// Mitsubishi GX Works2 project: BookEX6_34 DataProcess   PLC: Q13UDV

// global labels: Global
VAR_GLOBAL
  bVar0 AT M5000 : BOOL;
  abArray0 AT M5010 : ARRAY [0..49] OF BOOL;
  sStr0 AT D5000 : STRING[199];
  sStr1 AT D5100 : STRING[199];
  sStr2 AT D5200 : STRING[199];
  sStr3 AT D5300 : STRING[199];
  sStr4 AT D5400 : STRING[199];
  sStr5 AT D5500 : STRING[199];
  sStr6 AT D5600 : STRING[199];
  sStr7 AT D5700 : STRING[199];
  sStr8 AT D5800 : STRING[199];
  sStr9 AT D5900 : STRING[199];
  iVar0 AT D4500 : INT;
  iVar1 AT D4501 : INT;
  iVar2 AT D4502 : INT;
  iVar3 AT D4503 : INT;
  iVar4 AT D4504 : INT;
  iVar5 AT D4505 : INT;
  iVar6 AT D4506 : INT;
  iVar7 AT D4507 : INT;
  iVar8 AT D4508 : INT;
  iVar9 AT D4509 : INT;
  dVar0 AT D4510 : DINT;
  dVar1 AT D4512 : DINT;
  dVar2 AT D4514 : DINT;
  dVar3 AT D4516 : DINT;
  dVar4 AT D4518 : DINT;
  dVar5 AT D4520 : DINT;
  dVar6 AT D4522 : DINT;
  dVar7 AT D4524 : DINT;
  dVar8 AT D4526 : DINT;
  dVar9 AT D4528 : DINT;
  wVar0 AT D4530 : WORD;
  wVar1 AT D4531 : WORD;
  wVar2 AT D4532 : WORD;
  wVar3 AT D4533 : WORD;
  wVar4 AT D4534 : WORD;
  wVar5 AT D4535 : WORD;
  wVar6 AT D4536 : WORD;
  wVar7 AT D4537 : WORD;
  wVar8 AT D4538 : WORD;
  wVar9 AT D4539 : WORD;
  dwVar0 AT D4540 : DWORD;
  dwVar1 AT D4542 : DWORD;
  dwVar2 AT D4544 : DWORD;
  dwVar3 AT D4546 : DWORD;
  dwVar4 AT D4548 : DWORD;
  dwVar5 AT D4550 : DWORD;
  dwVar6 AT D4552 : DWORD;
  dwVar7 AT D4554 : DWORD;
  dwVar8 AT D4556 : DWORD;
  dwVar9 AT D4558 : DWORD;
  fsVar0 AT D4560 : REAL;
  fsVar1 AT D4562 : REAL;
  fsVar2 AT D4564 : REAL;
  fsVar3 AT D4566 : REAL;
  fsVar4 AT D4568 : REAL;
  fsVar5 AT D4570 : REAL;
  fsVar6 AT D4572 : REAL;
  fsVar7 AT D4574 : REAL;
  fsVar8 AT D4576 : REAL;
  fsVar9 AT D4578 : REAL;
  fdVar0 AT D4580 : LREAL;
  tTime0 AT D4620 : TIME;
  tTime1 AT D4622 : TIME;
  tTime2 AT D4624 : TIME;
  tTime3 AT D4626 : TIME;
  tTime4 AT D4628 : TIME;
  tTime5 AT D4630 : TIME;
  tTime6 AT D4632 : TIME;
  tTime7 AT D4634 : TIME;
  tTime8 AT D4636 : TIME;
  tTime9 AT D4638 : TIME;
  tTime10 AT D4640 : TIME;
  bVar1 AT M5001 : BOOL;
  bVar2 AT M5002 : BOOL;
  bVar3 AT M5003 : BOOL;
  bVar4 AT M5004 : BOOL;
  bVar5 AT M5005 : BOOL;
  bVar6 AT M5006 : BOOL;
  bVar7 AT M5007 : BOOL;
  bVar8 AT M5008 : BOOL;
  bVar9 AT M5009 : BOOL;
  abArray1 AT M5060 : ARRAY [0..49] OF BOOL;
  abArray2 AT M5110 : ARRAY [0..49] OF BOOL;
  abArray3 AT M5160 : ARRAY [0..49] OF BOOL;
  abArray4 AT M5210 : ARRAY [0..49] OF BOOL;
  abArray5 AT M5260 : ARRAY [0..49] OF BOOL;
  abArray6 AT M5310 : ARRAY [0..49] OF BOOL;
  abArray7 AT M5360 : ARRAY [0..49] OF BOOL;
  abArray8 AT M5410 : ARRAY [0..49] OF BOOL;
  abArray9 AT M5460 : ARRAY [0..49] OF BOOL;
  fdVar1 AT D4584 : LREAL;
  fdVar2 AT D4588 : LREAL;
  fdVar3 AT D4592 : LREAL;
  fdVar4 AT D4596 : LREAL;
  fdVar5 AT D4600 : LREAL;
  fdVar6 AT D4604 : LREAL;
  fdVar7 AT D4608 : LREAL;
  fdVar8 AT D4612 : LREAL;
  fdVar9 AT D4616 : LREAL;
  afsPen0 AT D2000 : ARRAY [0..499] OF REAL;
  afsPen1 AT D3000 : ARRAY [0..499] OF REAL;
END_VAR
// user libraries (not included): HMI

PROGRAM ExCCD
VAR
  aiVar8 : ARRAY [0..1] OF INT;
  aiVar16 : ARRAY [0..1] OF INT;
END_VAR
(* structured ladder/FBD written out as ST: instructions are called as NAME(EN, inputs, outputs); _pN, _eN, _tN stand for wires *)
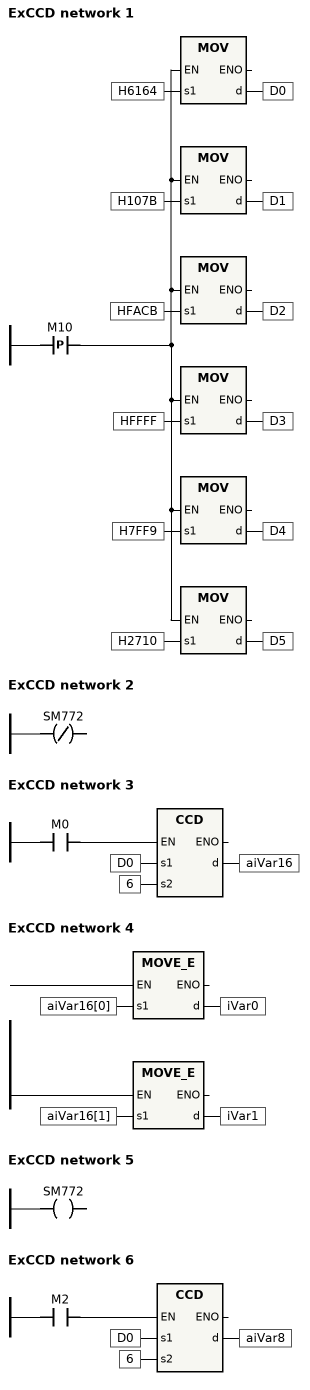
(* network 1 *)
_p1 := LDP(TRUE, M10);
MOV(_p1, H6164, D0);
MOV(_p1, H107B, D1);
MOV(_p1, HFACB, D2);
MOV(_p1, HFFFF, D3);
MOV(_p1, H7FF9, D4);
MOV(_p1, H2710, D5);
(* network 2 *)
SM772 := NOT TRUE;
(* network 3 *)
CCD(M0, D0, 6, aiVar16);
(* network 4 *)
MOVE_E(TRUE, aiVar16[0], iVar0);
MOVE_E(TRUE, aiVar16[1], iVar1);
(* network 5 *)
SM772 := TRUE;
(* network 6 *)
CCD(M2, D0, 6, aiVar8);
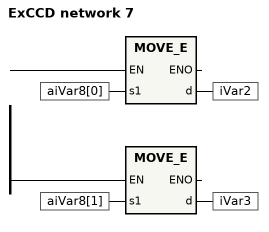
(* network 7 *)
MOVE_E(TRUE, aiVar8[0], iVar2);
MOVE_E(TRUE, aiVar8[1], iVar3);
END_PROGRAM

PROGRAM ExCRC
VAR
  aiVar0 : ARRAY [0..1] OF INT;
  aiVar1 : ARRAY [0..1] OF INT;
  aiVar2 : ARRAY [0..3] OF INT;
  aiVar3 : ARRAY [0..2] OF INT;
  Mov8INT_1 : Mov8INT;
  GetCRC_1 : GetCRC;
  GetCRC_2 : GetCRC;
END_VAR
(* structured ladder/FBD written out as ST: instructions are called as NAME(EN, inputs, outputs); _pN, _eN, _tN stand for wires *)
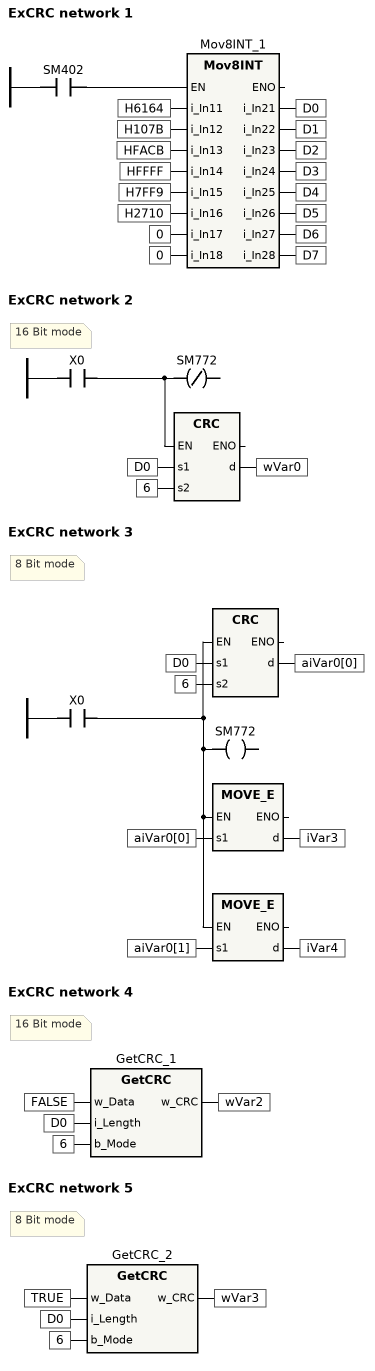
(* network 1 *)
Mov8INT_1(EN := SM402, i_In11 := H6164, i_In12 := H107B, i_In13 := HFACB, i_In14 := HFFFF, i_In15 := H7FF9, i_In16 := H2710, i_In17 := 0, i_In18 := 0, i_In21 => D0, i_In22 => D1, i_In23 => D2, i_In24 => D3, i_In25 => D4, i_In26 => D5, i_In27 => D6, i_In28 => D7);
(* network 2 *)
(* 16 Bit mode *)
SM772 := NOT X0;
CRC(X0, D0, 6, wVar0);
(* network 3 *)
(* 8 Bit mode *)
SM772 := X0;
CRC(X0, D0, 6, aiVar0[0]);
MOVE_E(X0, aiVar0[0], iVar3);
MOVE_E(X0, aiVar0[1], iVar4);
(* network 4 *)
(* 16 Bit mode *)
GetCRC_1(w_Data := FALSE, i_Length := D0, b_Mode := 6, w_CRC => wVar2);
(* network 5 *)
(* 8 Bit mode *)
GetCRC_2(w_Data := TRUE, i_Length := D0, b_Mode := 6, w_CRC => wVar3);
END_PROGRAM

PROGRAM ExDECO
VAR
  abArr0 : ARRAY [0..2] OF BOOL;
  Decode8_1 : Decode8;
  abArr1 : ARRAY [0..7] OF BOOL;
  Decode4_1 : Decode4;
  Decode8_2 : Decode8;
  bMan : BOOL;
  bSemi : BOOL;
  bAuto : BOOL;
  bMaint : BOOL;
END_VAR
(* structured ladder/FBD written out as ST: instructions are called as NAME(EN, inputs, outputs); _pN, _eN, _tN stand for wires *)
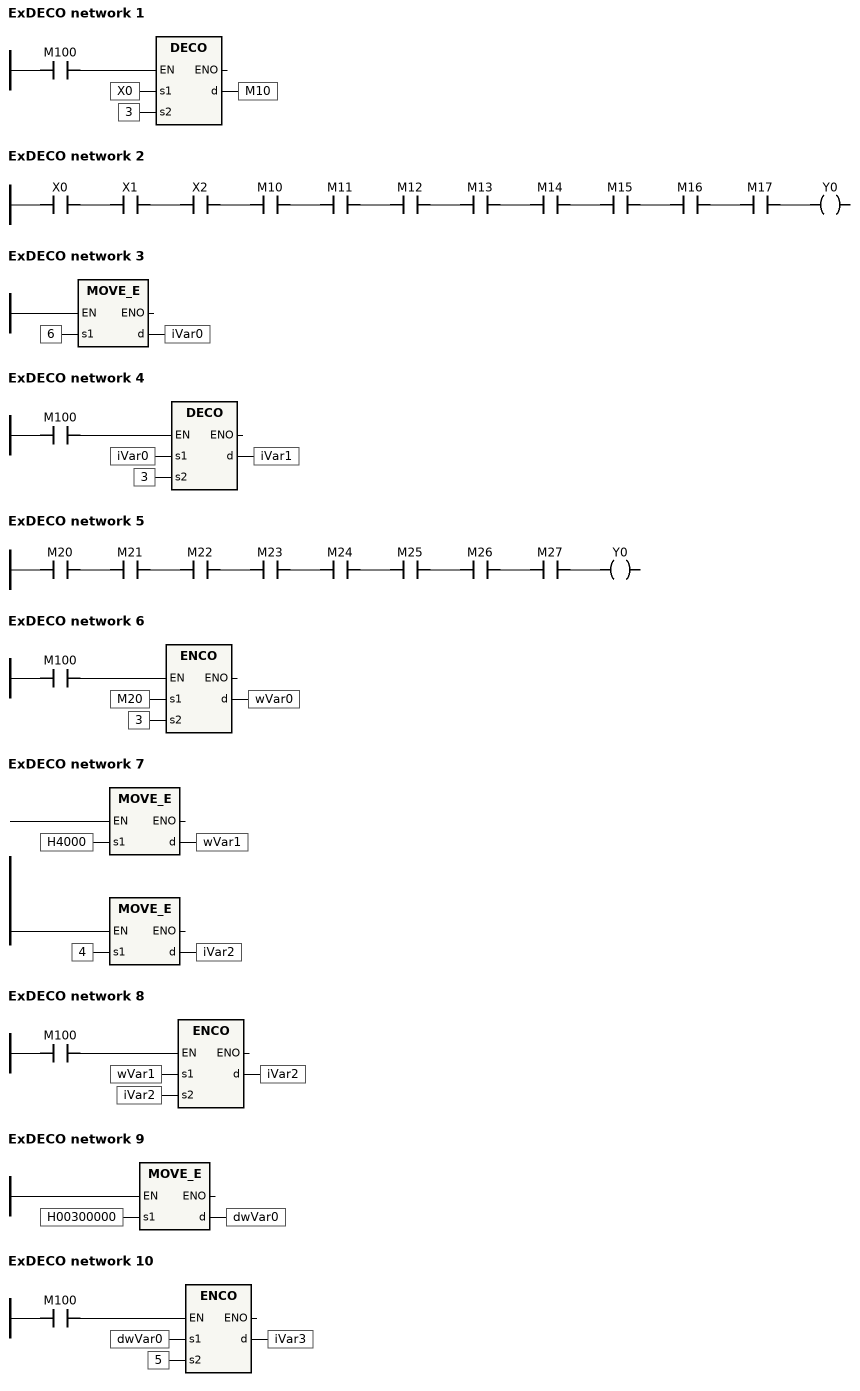
(* network 1 *)
DECO(M100, X0, 3, M10);
(* network 2 *)
Y0 := X0 AND X1 AND X2 AND M10 AND M11 AND M12 AND M13 AND M14 AND M15 AND M16 AND M17;
(* network 3 *)
MOVE_E(TRUE, 6, iVar0);
(* network 4 *)
DECO(M100, iVar0, 3, iVar1);
(* network 5 *)
Y0 := M20 AND M21 AND M22 AND M23 AND M24 AND M25 AND M26 AND M27;
(* network 6 *)
ENCO(M100, M20, 3, wVar0);
(* network 7 *)
MOVE_E(TRUE, H4000, wVar1);
MOVE_E(TRUE, 4, iVar2);
(* network 8 *)
ENCO(M100, wVar1, iVar2, iVar2);
(* network 9 *)
MOVE_E(TRUE, H00300000, dwVar0);
(* network 10 *)
ENCO(M100, dwVar0, 5, iVar3);
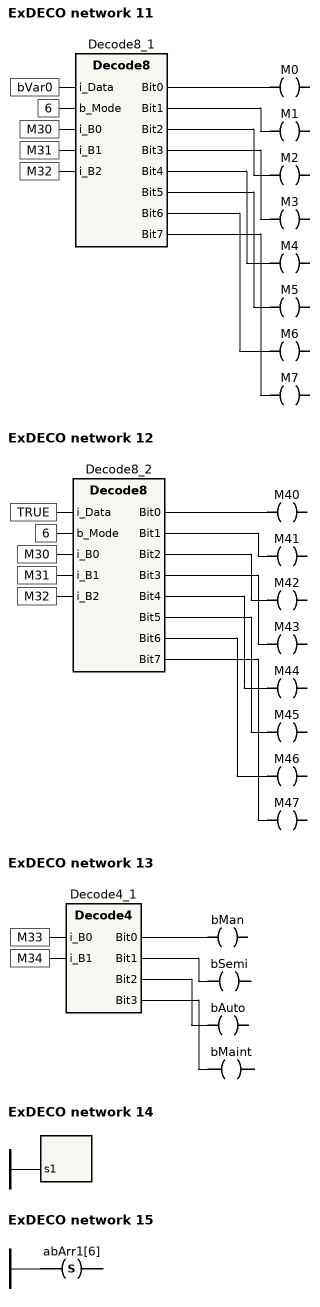
(* network 11 *)
Decode8_1(i_Data := bVar0, b_Mode := 6, i_B0 := M30, i_B1 := M31, i_B2 := M32);
M0 := Decode8_1.Bit0;
M1 := Decode8_1.Bit1;
M2 := Decode8_1.Bit2;
M3 := Decode8_1.Bit3;
M4 := Decode8_1.Bit4;
M5 := Decode8_1.Bit5;
M6 := Decode8_1.Bit6;
M7 := Decode8_1.Bit7;
(* network 12 *)
Decode8_2(i_Data := TRUE, b_Mode := 6, i_B0 := M30, i_B1 := M31, i_B2 := M32);
M40 := Decode8_2.Bit0;
M41 := Decode8_2.Bit1;
M42 := Decode8_2.Bit2;
M43 := Decode8_2.Bit3;
M44 := Decode8_2.Bit4;
M45 := Decode8_2.Bit5;
M46 := Decode8_2.Bit6;
M47 := Decode8_2.Bit7;
(* network 13 *)
Decode4_1(i_B0 := M33, i_B1 := M34);
bMan := Decode4_1.Bit0;
bSemi := Decode4_1.Bit1;
bAuto := Decode4_1.Bit2;
bMaint := Decode4_1.Bit3;
(* network 14 *)
(* element kind 10  <- TRUE *)
(* network 15 *)
SET(TRUE, abArr1[6]);
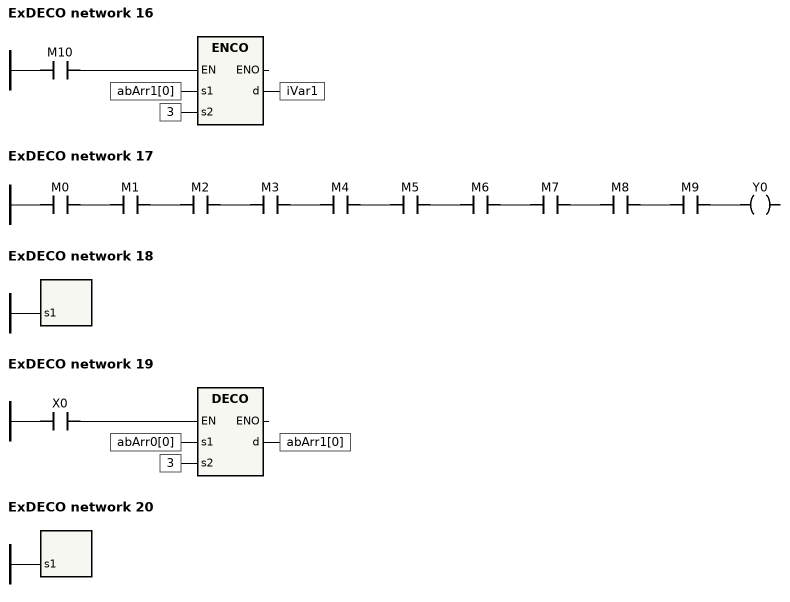
(* network 16 *)
ENCO(M10, abArr1[0], 3, iVar1);
(* network 17 *)
Y0 := M0 AND M1 AND M2 AND M3 AND M4 AND M5 AND M6 AND M7 AND M8 AND M9;
(* network 18 *)
(* element kind 10  <- TRUE *)
(* network 19 *)
DECO(X0, abArr0[0], 3, abArr1[0]);
(* network 20 *)
(* element kind 10  <- TRUE *)
END_PROGRAM

PROGRAM ExDIS
VAR
  Mov4WORD_1 : Mov4WORD;
  DDIS_1 : DDIS;
END_VAR
(* structured ladder/FBD written out as ST: instructions are called as NAME(EN, inputs, outputs); _pN, _eN, _tN stand for wires *)
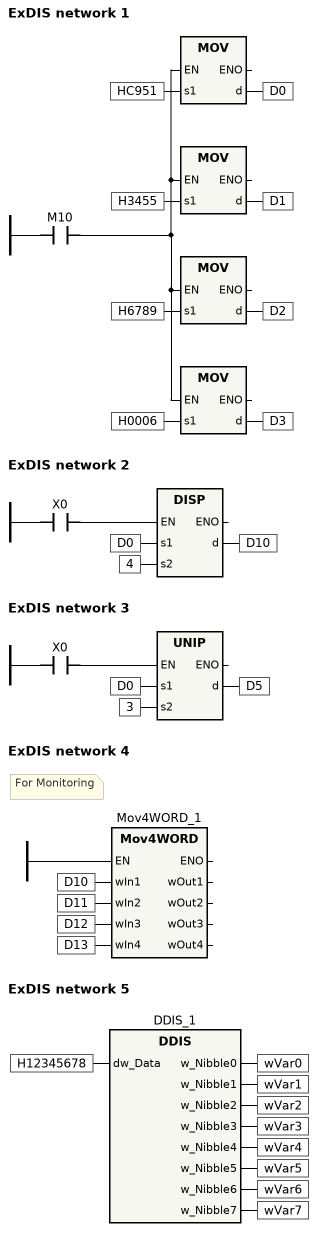
(* network 1 *)
MOV(M10, HC951, D0);
MOV(M10, H3455, D1);
MOV(M10, H6789, D2);
MOV(M10, H0006, D3);
(* network 2 *)
DISP(X0, D0, 4, D10);
(* network 3 *)
UNIP(X0, D0, 3, D5);
(* network 4 *)
(* For Monitoring *)
Mov4WORD_1(EN := TRUE, wIn1 := D10, wIn2 := D11, wIn3 := D12, wIn4 := D13);
(* network 5 *)
DDIS_1(dw_Data := H12345678, w_Nibble0 => wVar0, w_Nibble1 => wVar1, w_Nibble2 => wVar2, w_Nibble3 => wVar3, w_Nibble4 => wVar4, w_Nibble5 => wVar5, w_Nibble6 => wVar6, w_Nibble7 => wVar7);
END_PROGRAM

PROGRAM ExGetParity
VAR
  GetParity_1 : GetParity;
  awTestData : ARRAY [0..255] OF WORD;
  GetParity_2 : GetParity;
END_VAR
(* structured ladder/FBD written out as ST: instructions are called as NAME(EN, inputs, outputs); _pN, _eN, _tN stand for wires *)
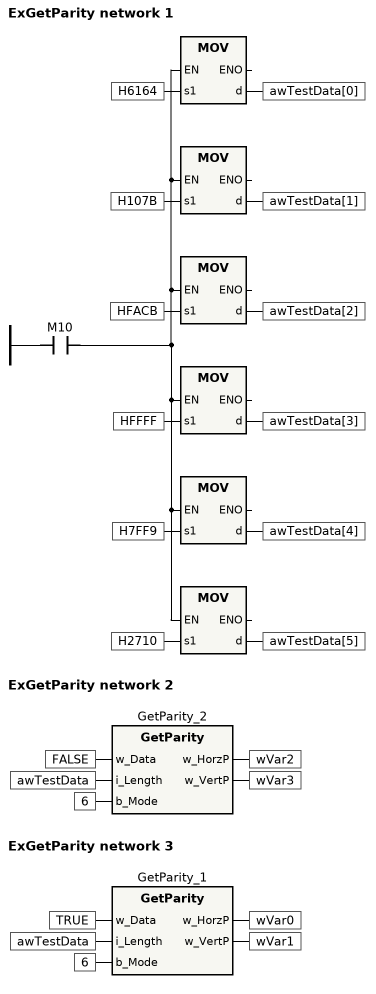
(* network 1 *)
MOV(M10, H6164, awTestData[0]);
MOV(M10, H107B, awTestData[1]);
MOV(M10, HFACB, awTestData[2]);
MOV(M10, HFFFF, awTestData[3]);
MOV(M10, H7FF9, awTestData[4]);
MOV(M10, H2710, awTestData[5]);
(* network 2 *)
GetParity_2(w_Data := FALSE, i_Length := awTestData, b_Mode := 6, w_HorzP => wVar2, w_VertP => wVar3);
(* network 3 *)
GetParity_1(w_Data := TRUE, i_Length := awTestData, b_Mode := 6, w_HorzP => wVar0, w_VertP => wVar1);
END_PROGRAM

PROGRAM ExMAX
VAR
  Mov4WORD_1 : Mov4WORD;
  Mov4WORD_2 : Mov4WORD;
  Mov4WORD_3 : Mov4WORD;
  dVa : ARRAY [0..1] OF DINT;
  RealMIN_MAX_1 : RealMIN_MAX;
  afsData : ARRAY [0..31] OF REAL;
END_VAR
(* structured ladder/FBD written out as ST: instructions are called as NAME(EN, inputs, outputs); _pN, _eN, _tN stand for wires *)
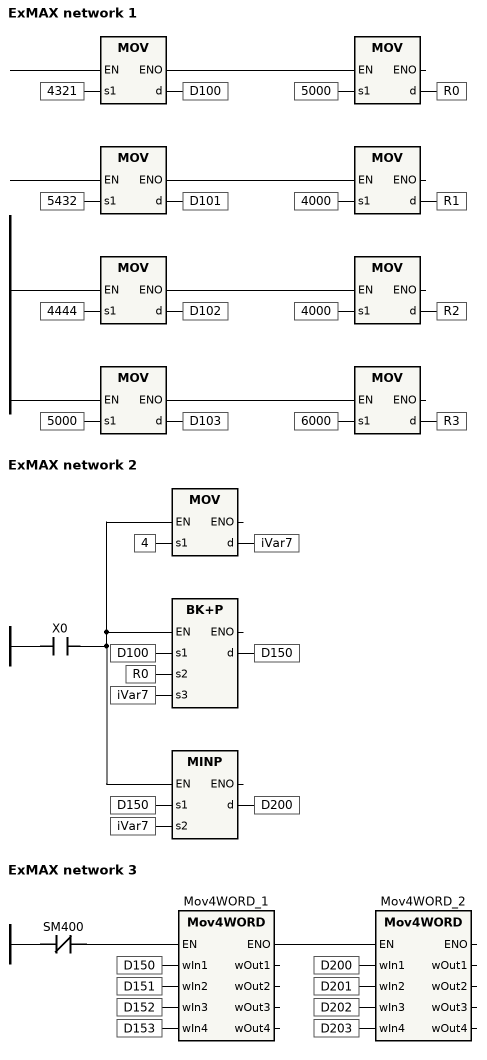
(* network 1 *)
_e1 := MOV(TRUE, 4321, D100);
MOV(_e1, 5000, R0);
_e2 := MOV(TRUE, 5432, D101);
MOV(_e2, 4000, R1);
_e3 := MOV(TRUE, 4444, D102);
MOV(_e3, 4000, R2);
_e4 := MOV(TRUE, 5000, D103);
MOV(_e4, 6000, R3);
(* network 2 *)
MOV(X0, 4, iVar7);
BK+P(X0, D100, R0, iVar7, D150);
MINP(X0, D150, iVar7, D200);
(* network 3 *)
Mov4WORD_1(EN := NOT SM400, wIn1 := D150, wIn2 := D151, wIn3 := D152, wIn4 := D153);
Mov4WORD_2(EN := Mov4WORD_1.ENO, wIn1 := D200, wIn2 := D201, wIn3 := D202, wIn4 := D203);
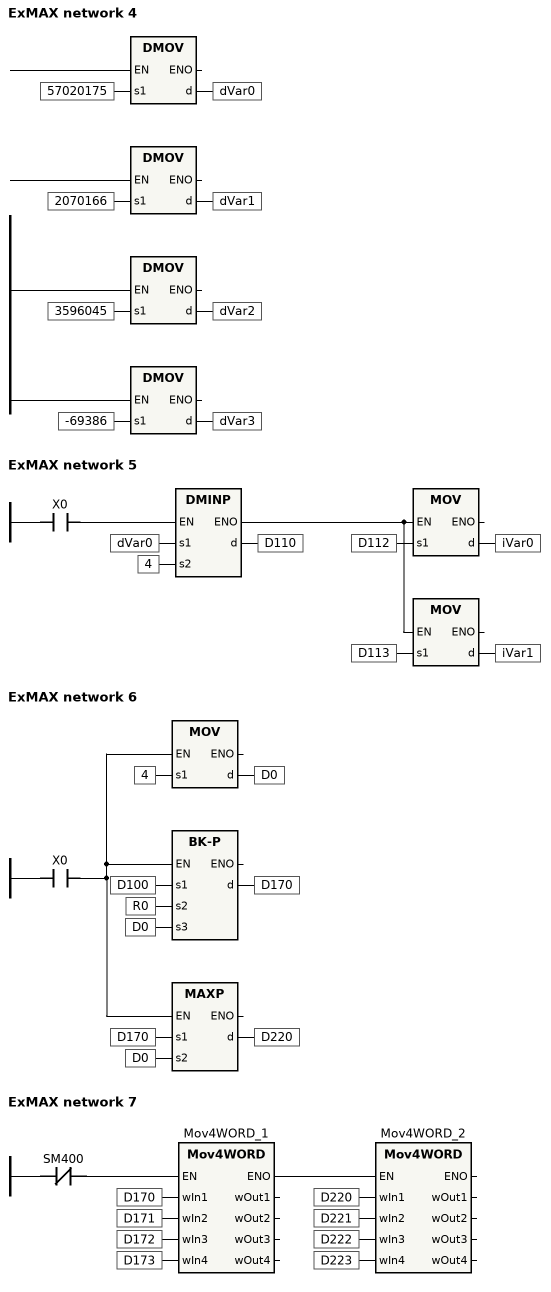
(* network 4 *)
DMOV(TRUE, 57020175, dVar0);
DMOV(TRUE, 2070166, dVar1);
DMOV(TRUE, 3596045, dVar2);
DMOV(TRUE, -69386, dVar3);
(* network 5 *)
_e1 := DMINP(X0, dVar0, 4, D110);
MOV(_e1, D112, iVar0);
MOV(_e1, D113, iVar1);
(* network 6 *)
MOV(X0, 4, D0);
BK-P(X0, D100, R0, D0, D170);
MAXP(X0, D170, D0, D220);
(* network 7 *)
Mov4WORD_1(EN := NOT SM400, wIn1 := D170, wIn2 := D171, wIn3 := D172, wIn4 := D173);
Mov4WORD_2(EN := Mov4WORD_1.ENO, wIn1 := D220, wIn2 := D221, wIn3 := D222, wIn4 := D223);
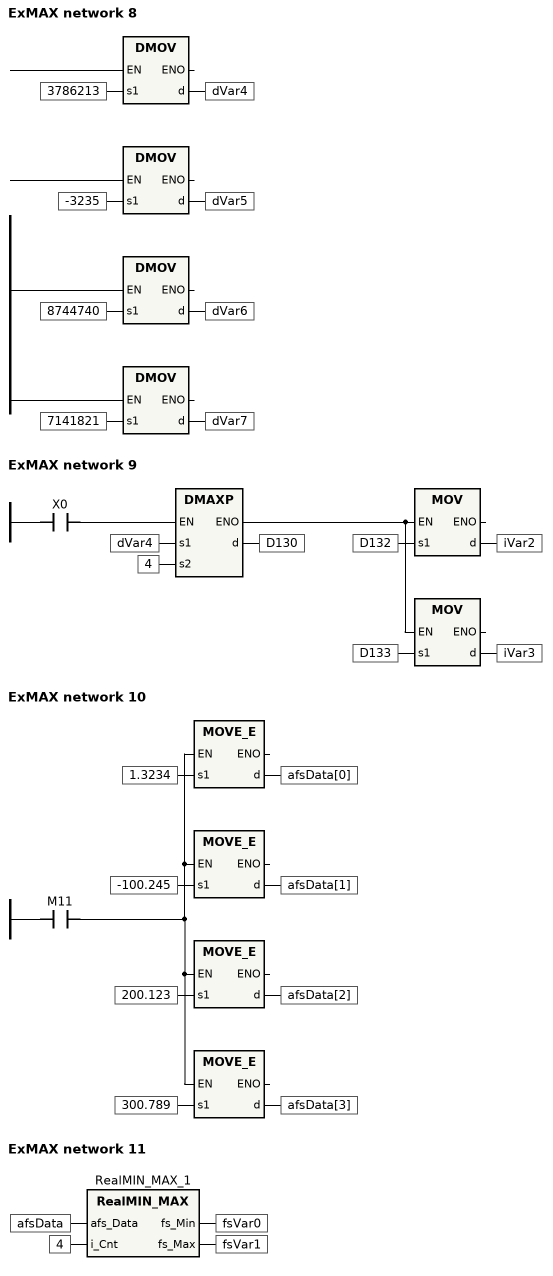
(* network 8 *)
DMOV(TRUE, 3786213, dVar4);
DMOV(TRUE, -3235, dVar5);
DMOV(TRUE, 8744740, dVar6);
DMOV(TRUE, 7141821, dVar7);
(* network 9 *)
_e1 := DMAXP(X0, dVar4, 4, D130);
MOV(_e1, D132, iVar2);
MOV(_e1, D133, iVar3);
(* network 10 *)
MOVE_E(M11, 1.3234, afsData[0]);
MOVE_E(M11, -100.245, afsData[1]);
MOVE_E(M11, 200.123, afsData[2]);
MOVE_E(M11, 300.789, afsData[3]);
(* network 11 *)
RealMIN_MAX_1(afs_Data := afsData, i_Cnt := 4, fs_Min => fsVar0, fs_Max => fsVar1);
END_PROGRAM

PROGRAM ExMEAN
VAR
  afsData : ARRAY [0..31] OF REAL;
END_VAR
(* structured ladder/FBD written out as ST: instructions are called as NAME(EN, inputs, outputs); _pN, _eN, _tN stand for wires *)
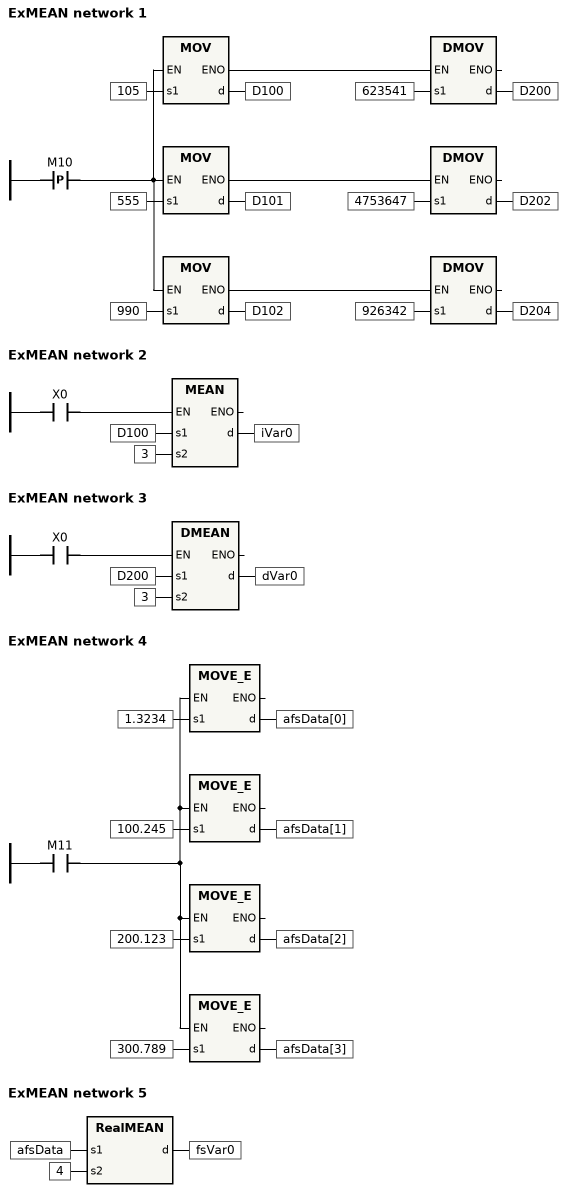
(* network 1 *)
_p1 := LDP(TRUE, M10);
_e2 := MOV(_p1, 105, D100);
DMOV(_e2, 623541, D200);
_e3 := MOV(_p1, 555, D101);
DMOV(_e3, 4753647, D202);
_e4 := MOV(_p1, 990, D102);
DMOV(_e4, 926342, D204);
(* network 2 *)
MEAN(X0, D100, 3, iVar0);
(* network 3 *)
DMEAN(X0, D200, 3, dVar0);
(* network 4 *)
MOVE_E(M11, 1.3234, afsData[0]);
MOVE_E(M11, 100.245, afsData[1]);
MOVE_E(M11, 200.123, afsData[2]);
MOVE_E(M11, 300.789, afsData[3]);
(* network 5 *)
fsVar0 := RealMEAN(afsData, 4);
END_PROGRAM

PROGRAM ExNDIS
VAR
  Mov4WORD_1 : Mov4WORD;
END_VAR
(* structured ladder/FBD written out as ST: instructions are called as NAME(EN, inputs, outputs); _pN, _eN, _tN stand for wires *)
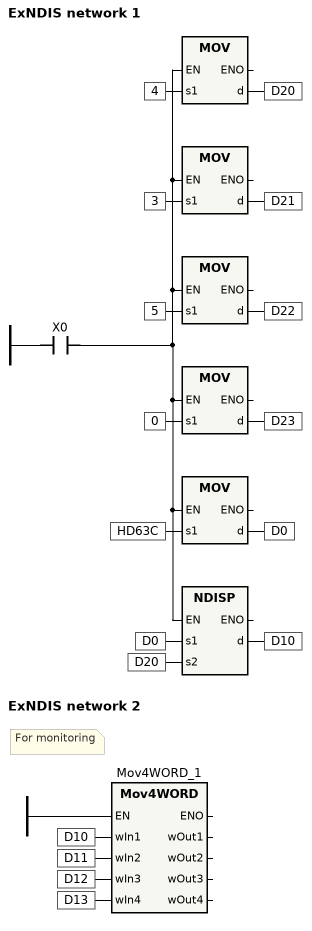
(* network 1 *)
MOV(X0, 4, D20);
MOV(X0, 3, D21);
MOV(X0, 5, D22);
MOV(X0, 0, D23);
MOV(X0, HD63C, D0);
NDISP(X0, D0, D20, D10);
(* network 2 *)
(* For monitoring *)
Mov4WORD_1(EN := TRUE, wIn1 := D10, wIn2 := D11, wIn3 := D12, wIn4 := D13);
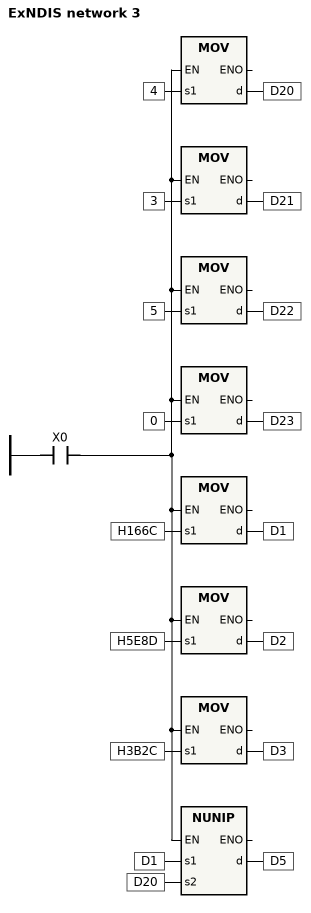
(* network 3 *)
MOV(X0, 4, D20);
MOV(X0, 3, D21);
MOV(X0, 5, D22);
MOV(X0, 0, D23);
MOV(X0, H166C, D1);
MOV(X0, H5E8D, D2);
MOV(X0, H3B2C, D3);
NUNIP(X0, D1, D20, D5);
END_PROGRAM

PROGRAM ExSearch
VAR
  Search_1 : Search;
  aiData : ARRAY [0..255] OF INT;
  DSearch_1 : DSearch;
  adData : ARRAY [0..255] OF DINT;
END_VAR
(* structured ladder/FBD written out as ST: instructions are called as NAME(EN, inputs, outputs); _pN, _eN, _tN stand for wires *)
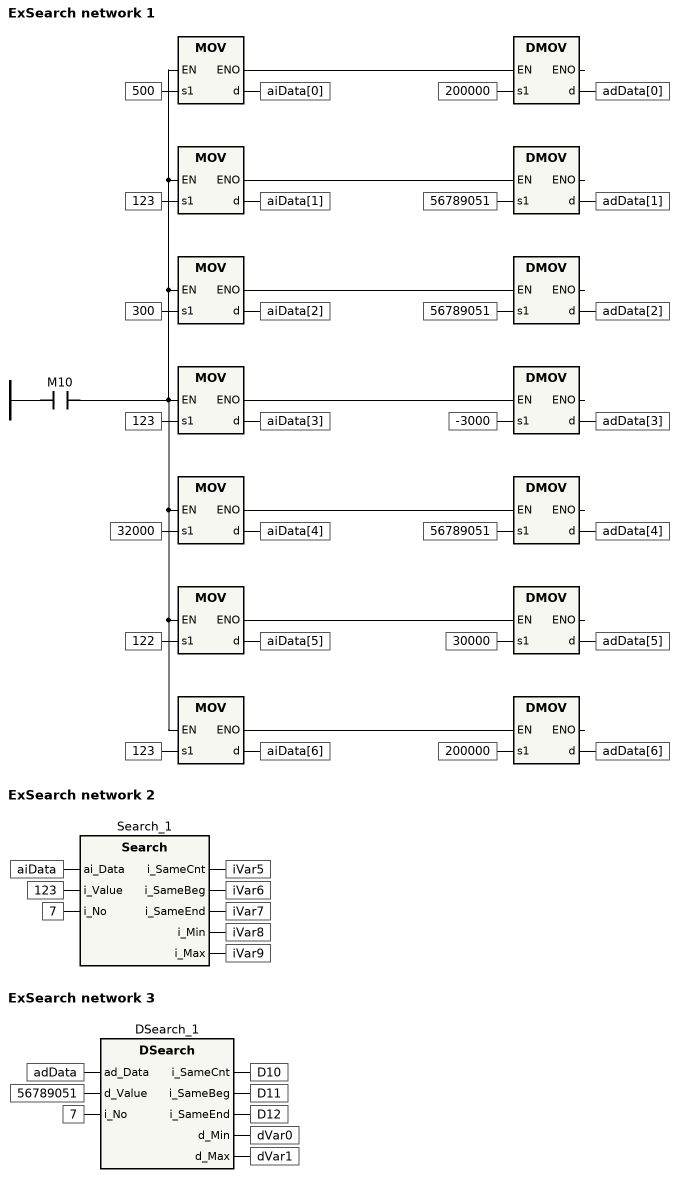
(* network 1 *)
_e1 := MOV(M10, 500, aiData[0]);
DMOV(_e1, 200000, adData[0]);
_e2 := MOV(M10, 123, aiData[1]);
DMOV(_e2, 56789051, adData[1]);
_e3 := MOV(M10, 300, aiData[2]);
DMOV(_e3, 56789051, adData[2]);
_e4 := MOV(M10, 123, aiData[3]);
DMOV(_e4, -3000, adData[3]);
_e5 := MOV(M10, 32000, aiData[4]);
DMOV(_e5, 56789051, adData[4]);
_e6 := MOV(M10, 122, aiData[5]);
DMOV(_e6, 30000, adData[5]);
_e7 := MOV(M10, 123, aiData[6]);
DMOV(_e7, 200000, adData[6]);
(* network 2 *)
Search_1(ai_Data := aiData, i_Value := 123, i_No := 7, i_SameCnt => iVar5, i_SameBeg => iVar6, i_SameEnd => iVar7, i_Min => iVar8, i_Max => iVar9);
(* network 3 *)
DSearch_1(ad_Data := adData, d_Value := 56789051, i_No := 7, i_SameCnt => D10, i_SameBeg => D11, i_SameEnd => D12, d_Min => dVar0, d_Max => dVar1);
END_PROGRAM

PROGRAM ExSEG
VAR
  aiClock : ARRAY [0..6] OF INT;
  aiMin : ARRAY [0..1] OF INT;
  aiSec : ARRAY [0..1] OF INT;
  aiHour : ARRAY [0..1] OF INT;
END_VAR
(* structured ladder/FBD written out as ST: instructions are called as NAME(EN, inputs, outputs); _pN, _eN, _tN stand for wires *)
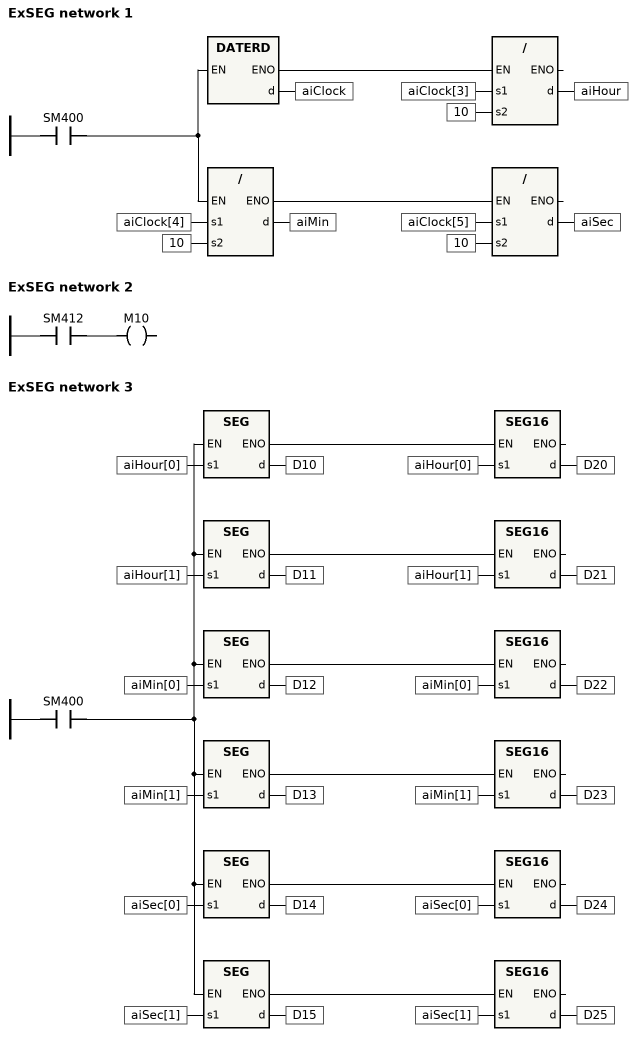
(* network 1 *)
_e1 := DATERD(SM400, aiClock);
/(_e1, aiClock[3], 10, aiHour);
_e2 := /(SM400, aiClock[4], 10, aiMin);
/(_e2, aiClock[5], 10, aiSec);
(* network 2 *)
M10 := SM412;
(* network 3 *)
_e1 := SEG(SM400, aiHour[0], D10);
SEG16(_e1, aiHour[0], D20);
_e2 := SEG(SM400, aiHour[1], D11);
SEG16(_e2, aiHour[1], D21);
_e3 := SEG(SM400, aiMin[0], D12);
SEG16(_e3, aiMin[0], D22);
_e4 := SEG(SM400, aiMin[1], D13);
SEG16(_e4, aiMin[1], D23);
_e5 := SEG(SM400, aiSec[0], D14);
SEG16(_e5, aiSec[0], D24);
_e6 := SEG(SM400, aiSec[1], D15);
SEG16(_e6, aiSec[1], D25);
END_PROGRAM

PROGRAM ExSER
VAR
  aiVar0 : ARRAY [0..1] OF INT;
  aiVar1 : ARRAY [0..1] OF INT;
  adVar0 : ARRAY [0..1] OF DINT;
  aiVar2 : ARRAY [0..3] OF INT;
  aiVar3 : ARRAY [0..2] OF INT;
END_VAR
(* structured ladder/FBD written out as ST: instructions are called as NAME(EN, inputs, outputs); _pN, _eN, _tN stand for wires *)
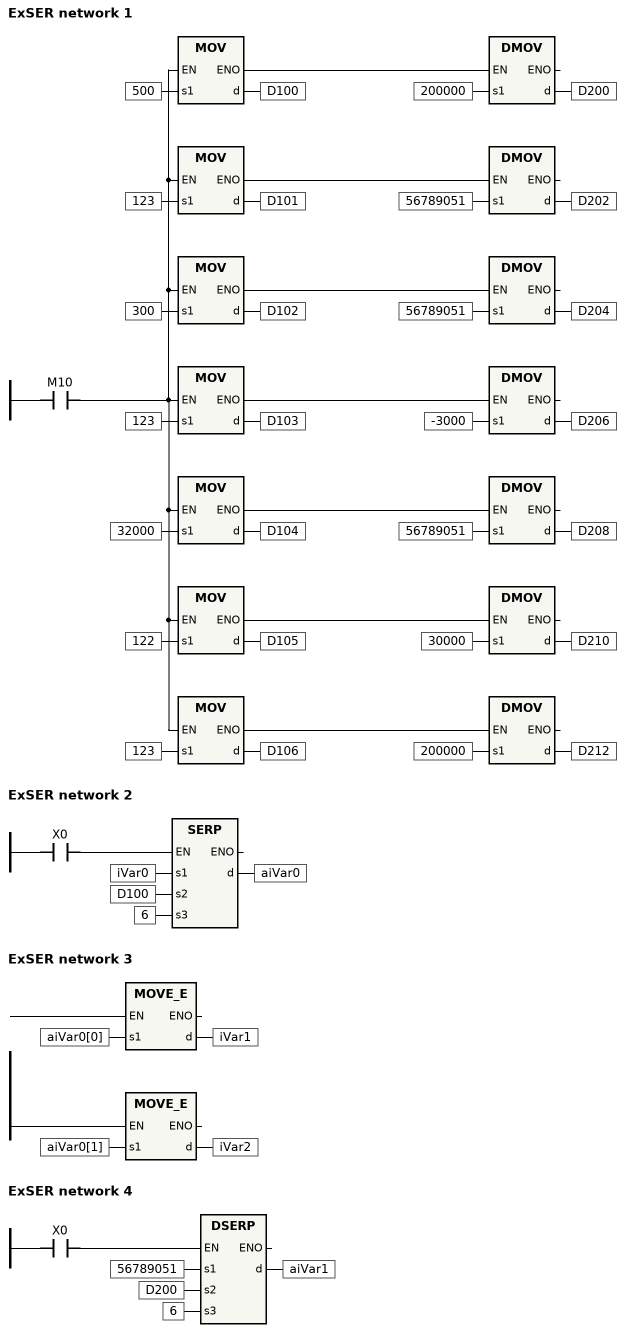
(* network 1 *)
_e1 := MOV(M10, 500, D100);
DMOV(_e1, 200000, D200);
_e2 := MOV(M10, 123, D101);
DMOV(_e2, 56789051, D202);
_e3 := MOV(M10, 300, D102);
DMOV(_e3, 56789051, D204);
_e4 := MOV(M10, 123, D103);
DMOV(_e4, -3000, D206);
_e5 := MOV(M10, 32000, D104);
DMOV(_e5, 56789051, D208);
_e6 := MOV(M10, 122, D105);
DMOV(_e6, 30000, D210);
_e7 := MOV(M10, 123, D106);
DMOV(_e7, 200000, D212);
(* network 2 *)
SERP(X0, iVar0, D100, 6, aiVar0);
(* network 3 *)
MOVE_E(TRUE, aiVar0[0], iVar1);
MOVE_E(TRUE, aiVar0[1], iVar2);
(* network 4 *)
DSERP(X0, 56789051, D200, 6, aiVar1);
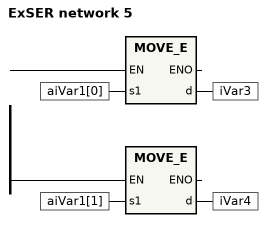
(* network 5 *)
MOVE_E(TRUE, aiVar1[0], iVar3);
MOVE_E(TRUE, aiVar1[1], iVar4);
END_PROGRAM

PROGRAM EXSORT
VAR
  SortBubble_1 : SortBubble;
  aiData300 : ARRAY [0..255] OF INT;
  SortSelection_1 : SortSelection;
  SortInsertion_1 : SortInsertion;
END_VAR
(* structured ladder/FBD written out as ST: instructions are called as NAME(EN, inputs, outputs); _pN, _eN, _tN stand for wires *)
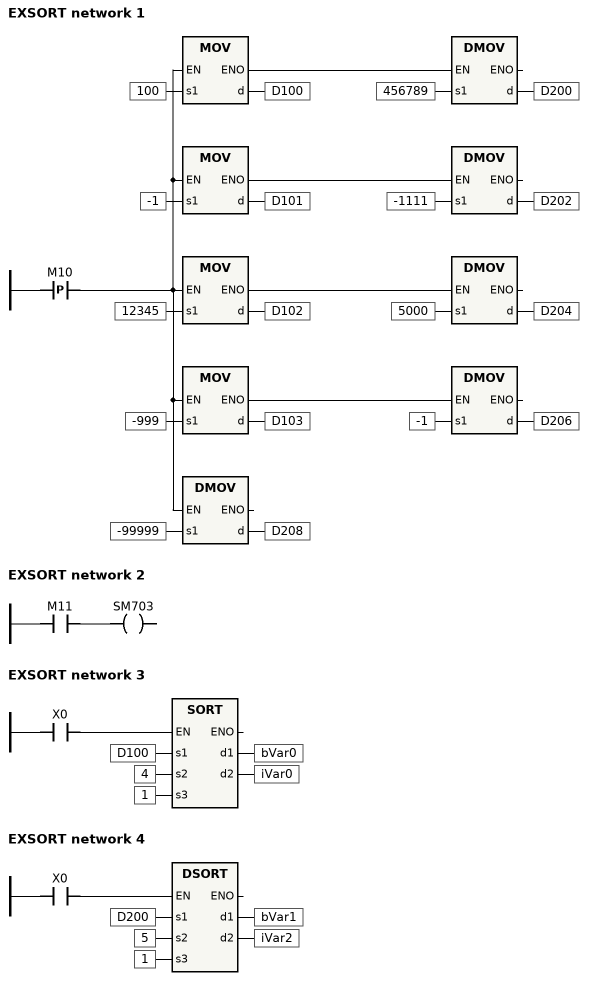
(* network 1 *)
_p1 := LDP(TRUE, M10);
_e2 := MOV(_p1, 100, D100);
DMOV(_e2, 456789, D200);
_e3 := MOV(_p1, -1, D101);
DMOV(_e3, -1111, D202);
_e4 := MOV(_p1, 12345, D102);
DMOV(_e4, 5000, D204);
_e5 := MOV(_p1, -999, D103);
DMOV(_e5, -1, D206);
DMOV(_p1, -99999, D208);
(* network 2 *)
SM703 := M11;
(* network 3 *)
SORT(X0, D100, 4, 1, bVar0, iVar0);
(* network 4 *)
DSORT(X0, D200, 5, 1, bVar1, iVar2);
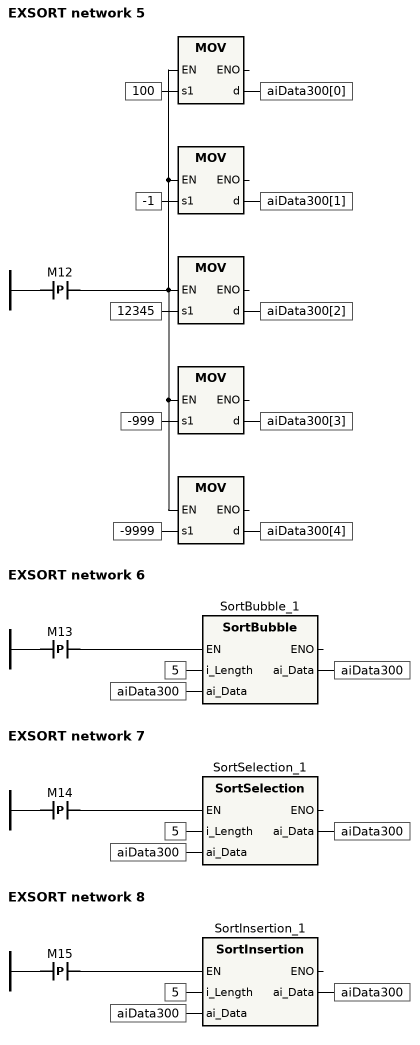
(* network 5 *)
_p1 := LDP(TRUE, M12);
MOV(_p1, 100, aiData300[0]);
MOV(_p1, -1, aiData300[1]);
MOV(_p1, 12345, aiData300[2]);
MOV(_p1, -999, aiData300[3]);
MOV(_p1, -9999, aiData300[4]);
(* network 6 *)
SortBubble_1(EN := LDP(TRUE, M13), i_Length := 5, ai_Data := aiData300);
aiData300 := SortBubble_1.ai_Data;
(* network 7 *)
SortSelection_1(EN := LDP(TRUE, M14), i_Length := 5, ai_Data := aiData300);
aiData300 := SortSelection_1.ai_Data;
(* network 8 *)
SortInsertion_1(EN := LDP(TRUE, M15), i_Length := 5, ai_Data := aiData300);
aiData300 := SortInsertion_1.ai_Data;
END_PROGRAM

PROGRAM ExSUM
(* structured ladder/FBD written out as ST: instructions are called as NAME(EN, inputs, outputs); _pN, _eN, _tN stand for wires *)
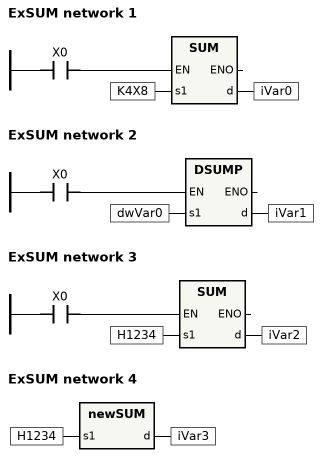
(* network 1 *)
SUM(X0, K4X8, iVar0);
(* network 2 *)
DSUMP(X0, dwVar0, iVar1);
(* network 3 *)
SUM(X0, H1234, iVar2);
(* network 4 *)
iVar3 := newSUM(H1234);
END_PROGRAM

PROGRAM ExWSUM
VAR
  aiVar0 : ARRAY [0..1] OF INT;
  aiVar1 : ARRAY [0..1] OF INT;
  adVar0 : ARRAY [0..1] OF DINT;
  aiVar2 : ARRAY [0..3] OF INT;
  aiVar3 : ARRAY [0..2] OF INT;
END_VAR
(* structured ladder/FBD written out as ST: instructions are called as NAME(EN, inputs, outputs); _pN, _eN, _tN stand for wires *)
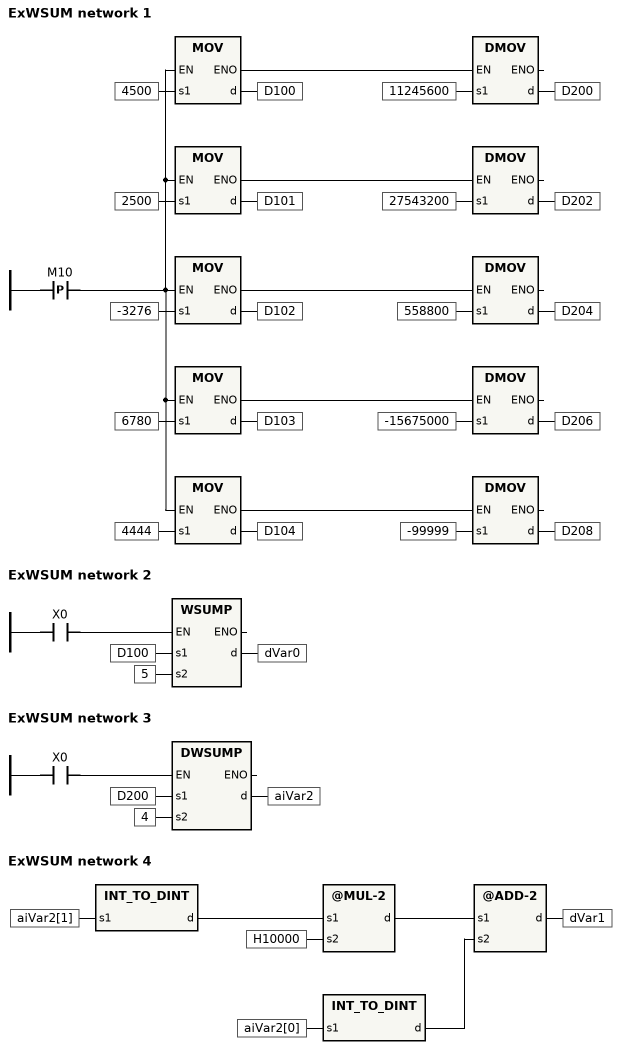
(* network 1 *)
_p1 := LDP(TRUE, M10);
_e2 := MOV(_p1, 4500, D100);
DMOV(_e2, 11245600, D200);
_e3 := MOV(_p1, 2500, D101);
DMOV(_e3, 27543200, D202);
_e4 := MOV(_p1, -3276, D102);
DMOV(_e4, 558800, D204);
_e5 := MOV(_p1, 6780, D103);
DMOV(_e5, -15675000, D206);
_e6 := MOV(_p1, 4444, D104);
DMOV(_e6, -99999, D208);
(* network 2 *)
WSUMP(X0, D100, 5, dVar0);
(* network 3 *)
DWSUMP(X0, D200, 4, aiVar2);
(* network 4 *)
dVar1 := @ADD-2(@MUL-2(INT_TO_DINT(aiVar2[1]), H10000), INT_TO_DINT(aiVar2[0]));
END_PROGRAM

PROGRAM ExWTOB
VAR
  Mov4WORD_1 : Mov4WORD;
  Mov8WORD_1 : Mov8WORD;
  Mov8WORD_2 : Mov8WORD;
  Mov4WORD_2 : Mov4WORD;
  ConvIP2Byte_1 : ConvIP2Byte;
  Mov4WORD_3 : Mov4WORD;
  Mov4WORD_4 : Mov4WORD;
  newWTOB_1 : newWTOB;
  Mov4WORD_5 : Mov4WORD;
  Mov4WORD_6 : Mov4WORD;
  Mov4WORD_7 : Mov4WORD;
END_VAR
(* structured ladder/FBD written out as ST: instructions are called as NAME(EN, inputs, outputs); _pN, _eN, _tN stand for wires *)
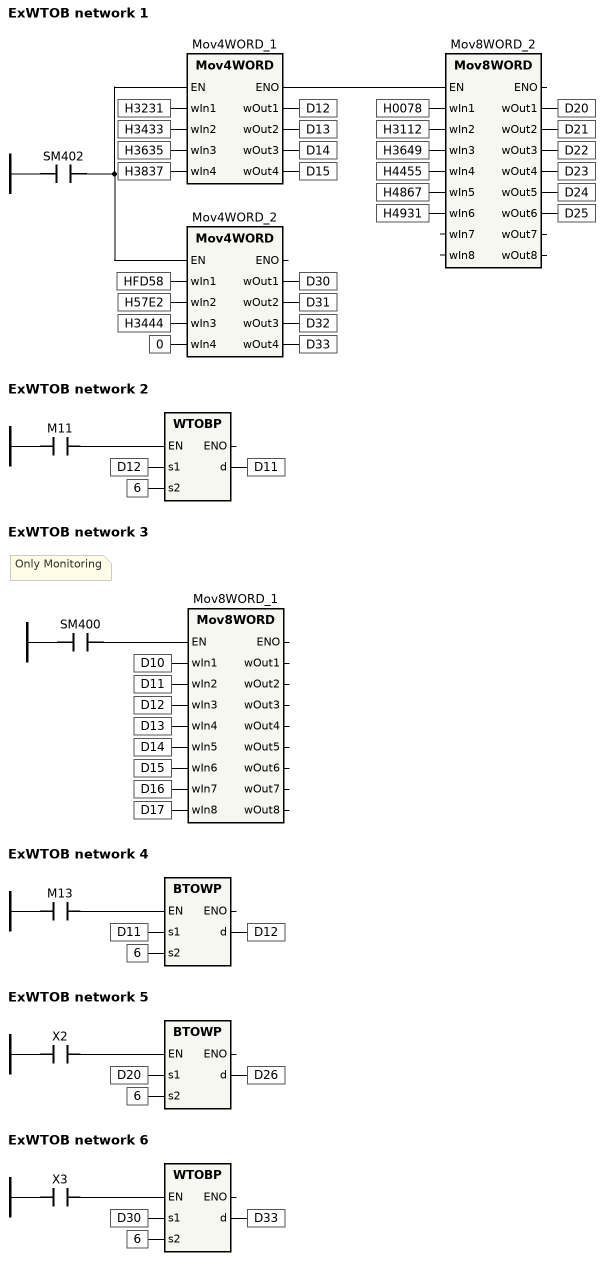
(* network 1 *)
Mov4WORD_1(EN := SM402, wIn1 := H3231, wIn2 := H3433, wIn3 := H3635, wIn4 := H3837, wOut1 => D12, wOut2 => D13, wOut3 => D14, wOut4 => D15);
Mov8WORD_2(EN := Mov4WORD_1.ENO, wIn1 := H0078, wIn2 := H3112, wIn3 := H3649, wIn4 := H4455, wIn5 := H4867, wIn6 := H4931, wOut1 => D20, wOut2 => D21, wOut3 => D22, wOut4 => D23, wOut5 => D24, wOut6 => D25);
Mov4WORD_2(EN := SM402, wIn1 := HFD58, wIn2 := H57E2, wIn3 := H3444, wIn4 := 0, wOut1 => D30, wOut2 => D31, wOut3 => D32, wOut4 => D33);
(* network 2 *)
WTOBP(M11, D12, 6, D11);
(* network 3 *)
(* Only Monitoring *)
Mov8WORD_1(EN := SM400, wIn1 := D10, wIn2 := D11, wIn3 := D12, wIn4 := D13, wIn5 := D14, wIn6 := D15, wIn7 := D16, wIn8 := D17);
(* network 4 *)
BTOWP(M13, D11, 6, D12);
(* network 5 *)
BTOWP(X2, D20, 6, D26);
(* network 6 *)
WTOBP(X3, D30, 6, D33);
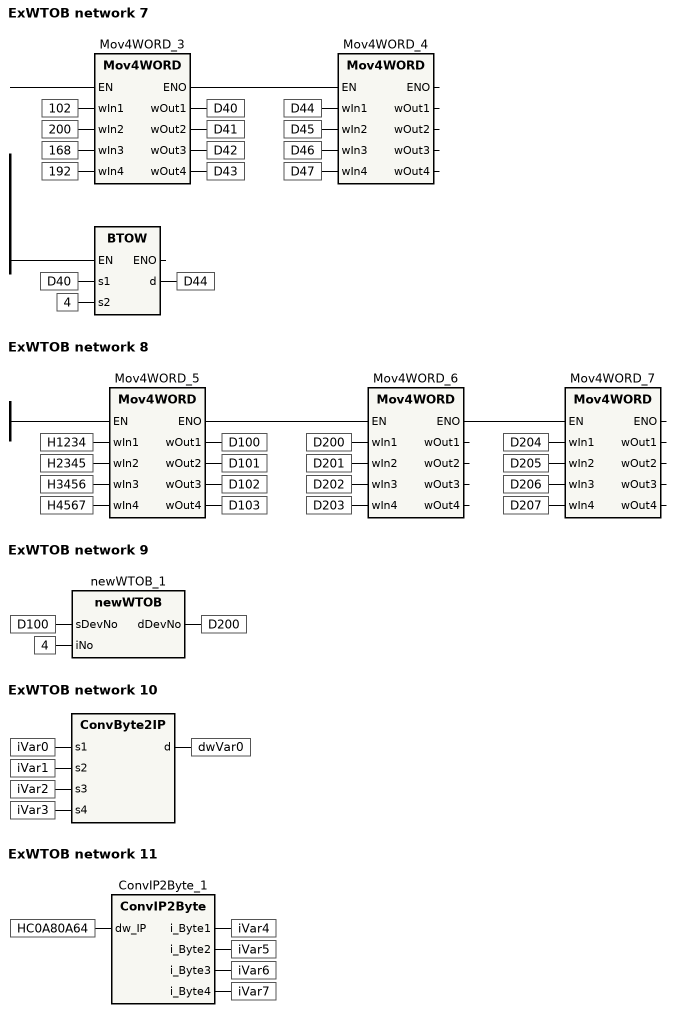
(* network 7 *)
Mov4WORD_3(EN := TRUE, wIn1 := 102, wIn2 := 200, wIn3 := 168, wIn4 := 192, wOut1 => D40, wOut2 => D41, wOut3 => D42, wOut4 => D43);
Mov4WORD_4(EN := Mov4WORD_3.ENO, wIn1 := D44, wIn2 := D45, wIn3 := D46, wIn4 := D47);
BTOW(TRUE, D40, 4, D44);
(* network 8 *)
Mov4WORD_5(EN := TRUE, wIn1 := H1234, wIn2 := H2345, wIn3 := H3456, wIn4 := H4567, wOut1 => D100, wOut2 => D101, wOut3 => D102, wOut4 => D103);
Mov4WORD_6(EN := Mov4WORD_5.ENO, wIn1 := D200, wIn2 := D201, wIn3 := D202, wIn4 := D203);
Mov4WORD_7(EN := Mov4WORD_6.ENO, wIn1 := D204, wIn2 := D205, wIn3 := D206, wIn4 := D207);
(* network 9 *)
newWTOB_1(sDevNo := D100, iNo := 4, dDevNo => D200);
(* network 10 *)
dwVar0 := ConvByte2IP(iVar0, iVar1, iVar2, iVar3);
(* network 11 *)
ConvIP2Byte_1(dw_IP := HC0A80A64, i_Byte1 => iVar4, i_Byte2 => iVar5, i_Byte3 => iVar6, i_Byte4 => iVar7);
END_PROGRAM

FUNCTION_BLOCK DDIS
VAR_INPUT
  dw_Data : DWORD;
END_VAR
VAR_OUTPUT
  w_Nibble0 : WORD;
  w_Nibble1 : WORD;
  w_Nibble2 : WORD;
  w_Nibble3 : WORD;
  w_Nibble4 : WORD;
  w_Nibble5 : WORD;
  w_Nibble6 : WORD;
  w_Nibble7 : WORD;
END_VAR
VAR
  dwx : DWORD;
END_VAR
;
dwx := dw_Data;
w_Nibble0 := DWORD_TO_WORD(dwx AND H0000000F);
DROR(TRUE, 4, dwx) ;
w_Nibble1 := DWORD_TO_WORD(dwx AND H0000000F);
DROR(TRUE, 4, dwx) ;
w_Nibble2 := DWORD_TO_WORD(dwx AND H0000000F);
DROR(TRUE, 4, dwx) ;
w_Nibble3 := DWORD_TO_WORD(dwx AND H0000000F);
DROR(TRUE, 4, dwx) ;
w_Nibble4 := DWORD_TO_WORD(dwx AND H0000000F);
DROR(TRUE, 4, dwx) ;
w_Nibble5 := DWORD_TO_WORD(dwx AND H0000000F);
DROR(TRUE, 4, dwx) ;
w_Nibble6 := DWORD_TO_WORD(dwx AND H0000000F);
DROR(TRUE, 4, dwx) ;
w_Nibble7 := DWORD_TO_WORD(dwx AND H0000000F);
END_FUNCTION_BLOCK

FUNCTION_BLOCK Decode4
VAR_OUTPUT
  Bit0 : BOOL;
  Bit1 : BOOL;
  Bit2 : BOOL;
  Bit3 : BOOL;
END_VAR
VAR_INPUT
  i_B0 : BOOL;
  i_B1 : BOOL;
END_VAR
;
Bit0 := NOT i_B0 AND NOT i_B1;
Bit1 := i_B0 AND NOT i_B1;
Bit2 := NOT i_B0 AND i_B1;
Bit3 := i_B0 AND i_B1;
END_FUNCTION_BLOCK

FUNCTION_BLOCK Decode8
VAR_INPUT
  i_Data : INT;
END_VAR
VAR_OUTPUT
  Bit0 : BOOL;
  Bit1 : BOOL;
  Bit2 : BOOL;
  Bit3 : BOOL;
  Bit4 : BOOL;
  Bit5 : BOOL;
  Bit6 : BOOL;
  Bit7 : BOOL;
END_VAR
VAR
  ix : INT;
END_VAR
VAR_INPUT
  b_Mode : BOOL;
  i_B0 : BOOL;
  i_B1 : BOOL;
  i_B2 : BOOL;
END_VAR
;
IF b_Mode THEN
	ix := BOOL_TO_INT(i_B0)+BOOL_TO_INT(i_B1)*2+BOOL_TO_INT(i_B2)*4;
ELSE
	ix := i_Data MOD 8;
END_IF;
Bit0 := FALSE;
Bit1 := FALSE;
Bit2 := FALSE;
Bit3 := FALSE;
Bit4 := FALSE;
Bit5 := FALSE;
Bit6 := FALSE;
Bit7 := FALSE;

CASE ix OF
	0 : Bit0 := TRUE;
	1 : Bit1 := TRUE;
	2 : Bit2 := TRUE;
	3 : Bit3 := TRUE;
	4 : Bit4 := TRUE;
	5 : Bit5 := TRUE;
	6 : Bit6 := TRUE;
	7 : Bit7 := TRUE;
END_CASE;
END_FUNCTION_BLOCK

FUNCTION_BLOCK DSearch
VAR_INPUT
  ad_Data : ARRAY [0..255] OF DINT;
  d_Value : DINT;
  i_No : INT;
END_VAR
VAR_OUTPUT
  i_SameCnt : INT;
  i_SameBeg : INT;
  i_SameEnd : INT;
  d_Min : DINT;
  d_Max : DINT;
END_VAR
VAR
  ix : INT;
  dVar : DINT;
  bFound : BOOL;
END_VAR
;
i_SameCnt 		:= 0;
i_SameBeg 	:= 0;
i_SameEnd 	:= 0;
d_Min 				:= H7FFFFFFF;
d_Max 				:= H80000000;
bFound 			:= FALSE;

FOR ix := 0 TO i_No-1 DO 
	dVar := ad_Data[ix];
	IF dVar = d_Value THEN
		i_SameCnt := i_SameCnt + 1;
		IF NOT bFound THEN
			i_SameBeg := ix + 1;
			bFound := TRUE;
		END_IF;
		i_SameEnd := ix + 1;
	END_IF;	
	IF d_Min > dVar THEN
		d_Min := dVar;
	END_IF;
	IF d_Max < dVar THEN
		d_Max := dVar;
	END_IF;
END_FOR;
END_FUNCTION_BLOCK

FUNCTION_BLOCK GetCRC
VAR_INPUT
  w_Data : WORD;
  i_Length : INT;
END_VAR
VAR_OUTPUT
  w_CRC : WORD;
END_VAR
VAR_INPUT
  b_Mode : BOOL;
END_VAR
VAR
  ix : INT;
  wCRC : WORD;
  wx : WORD;
  wLow : WORD;
  wHigh : WORD;
  iLeng : INT;
  wBuff : ARRAY [0..255] OF WORD;
  iy : INT;
  wBuff_org : ARRAY [0..255] OF WORD;
END_VAR
;	
BMOV(TRUE, w_Data, i_Length, wBuff_org[0]); 
IF b_Mode THEN
	(* 8Bit Mode *)
	FOR ix := 0 TO i_Length-1 DO 
		wBuff[ix] := wBuff_org[ix] AND H00FF;
	END_FOR;
ELSE
	(* 16 Bit Mode *)
	iy := 0;
	FOR ix := 0 TO (i_Length-1)/2 DO 
		wBuff[iy] := wBuff_org[ix] AND H00FF;
		wx := wBuff_org[ix];
		SWAP(TRUE, wx);
		wBuff[iy+1] := wx AND H00FF;
		iy := iy+2;
	END_FOR;
END_IF;	

wCRC := HFFFF;
FOR ix := 0 TO i_Length-1 DO 
	wCRC := wCRC XOR wBuff[ix]; 
	FOR iy := 0 TO 7 DO 
		SFR(TRUE, 1, wCRC);
		IF SM700 THEN
			wCRC := wCRC XOR HA001;
		END_IF;
	END_FOR;
END_FOR;

w_CRC := wCRC;
END_FUNCTION_BLOCK

FUNCTION_BLOCK GetParity
VAR_INPUT
  w_Data : ARRAY [0..255] OF WORD;
  i_Length : INT;
END_VAR
VAR_OUTPUT
  w_HorzP : WORD;
  w_VertP : WORD;
END_VAR
VAR_INPUT
  b_Mode : BOOL;
END_VAR
VAR
  ix : INT;
  iSum : INT;
  wHoriz : WORD;
  wLow : WORD;
  wHigh : WORD;
  iLeng : INT;
  wBuff : ARRAY [0..255] OF WORD;
  iy : INT;
END_VAR
;
IF b_Mode THEN
	(* 8Bit Mode *)
	FOR ix := 0 TO i_Length-1 DO 
		wBuff[ix] := w_Data[ix] AND H00FF;
	END_FOR;
ELSE
	(* 16 Bit Mode *)
	iy := 0;
	FOR ix := 0 TO (i_Length/2)-1 DO 
		wBuff[iy] := w_Data[ix] AND H00FF;
		wHoriz := w_Data[ix];
		SWAP(TRUE, wHoriz);
		wBuff[iy+1] := wHoriz AND H00FF;
		iy := iy+2;
	END_FOR;
END_IF;	

iSum := 0;
wHoriz := 0;
FOR ix := 0 TO i_Length-1 DO 
	iSum := iSum + WORD_TO_INT(wBuff[ix]);
	wHoriz := wHoriz XOR wBuff[ix];
END_FOR;

w_VertP := INT_TO_WORD(iSum);
w_HorzP := wHoriz;
END_FUNCTION_BLOCK

FUNCTION RealMEAN
VAR_INPUT
  afs_Data : ARRAY [0..31] OF REAL;
  i_Cnt : INT;
END_VAR
VAR
  ix : INT;
  fdReal : LREAL;
END_VAR
;
IF i_Cnt = 0 OR i_Cnt > 31 THEN
	RETURN;
END_IF;
FdReal := 0.0;
FOR ix := 0 TO i_Cnt -1 DO 
	fdReal := fdReal + REAL_TO_LREAL(afs_Data[ix]);
END_FOR;
RealMEAN := LREAL_TO_REAL(fdReal / INT_TO_LREAL(ix));
END_FUNCTION

FUNCTION_BLOCK RealMIN_MAX
VAR_INPUT
  afs_Data : ARRAY [0..31] OF REAL;
  i_Cnt : INT;
END_VAR
VAR
  ix : INT;
  minReal : REAL;
END_VAR
VAR_OUTPUT
  fs_Min : REAL;
  fs_Max : REAL;
END_VAR
VAR
  maxReal : REAL;
END_VAR
;
IF i_Cnt = 0 OR i_Cnt > 31 THEN
	RETURN;
END_IF;
minReal := 0.0;
maxReal := 0.0;
FOR ix := 0 TO i_Cnt -1 DO 
	IF minReal > afs_Data[ix] THEN
		minReal := afs_Data[ix];
	END_IF;
	IF maxReal < afs_Data[ix] THEN
		maxReal := afs_Data[ix];
	END_IF;
END_FOR;

fs_Max := maxReal;
fs_Min := minReal;
END_FUNCTION_BLOCK

FUNCTION_BLOCK Search
VAR_INPUT
  ai_Data : ARRAY [0..255] OF INT;
  i_Value : INT;
  i_No : INT;
END_VAR
VAR_OUTPUT
  i_SameCnt : INT;
  i_SameBeg : INT;
  i_SameEnd : INT;
  i_Min : INT;
  i_Max : INT;
END_VAR
VAR
  ix : INT;
  iy : INT;
  iz : INT;
  bFound : BOOL;
END_VAR
;
i_SameCnt 		:= 0;
i_SameBeg 	:= 0;
i_SameEnd 	:= 0;
i_Min 					:= H7FFF;
i_Max 				:= H8000;
bFound 			:= FALSE;

FOR ix := 0 TO i_No-1 DO 
	iy := ai_Data[ix];
	IF iy = i_Value THEN
		i_SameCnt := i_SameCnt + 1;
		IF NOT bFound THEN
			i_SameBeg := ix + 1;
			bFound := TRUE;
		END_IF;
		i_SameEnd := ix + 1;
	END_IF;
	IF i_Min > iy THEN
		i_Min := iy;
	END_IF;
	IF i_Max < iy THEN
		i_Max := iy;
	END_IF;
END_FOR;
END_FUNCTION_BLOCK

FUNCTION SEG16
VAR_INPUT
  i_Data : INT;
END_VAR
VAR
  Temp : WORD;
END_VAR
;
CASE i_Data MOD 16 OF
	0 :	Temp := H90FF;
	1 :	Temp := H100C;
	2 :	Temp := H0377;
	3 :	Temp := H023F;
	4 :	Temp := H038C;
	5 :	Temp := H03BB;
	6 :	Temp := H03FB;
	7 :	Temp := H000F;
	8 :	Temp := H03FF;
	9 :	Temp := H03BF;
	10 :	Temp := H03CF;
	11 :	Temp := H4A3F;
	12 :	Temp := H00F3;
	13 :	Temp := H483F;
	14 :	Temp := H01F3;
	15 :	Temp := H01C3;
END_CASE;
SEG16 := Temp;
END_FUNCTION

FUNCTION_BLOCK SortBubble
VAR_INPUT
  i_Length : INT;
END_VAR
VAR
  ix : INT;
  iy : INT;
  iz : INT;
END_VAR
VAR_IN_OUT
  ai_Data : ARRAY [0..255] OF INT;
END_VAR
;
FOR ix := 0 TO i_Length-2 DO 
	FOR iy := 0 TO i_Length-2 DO 
		IF ai_Data[iy] > ai_Data[iy+1] THEN
			iz := ai_Data[iy];
			ai_Data[iy] := ai_Data[iy+1];
			ai_Data[iy+1] := iz;
		END_IF;
	END_FOR;
END_FOR;
END_FUNCTION_BLOCK

FUNCTION_BLOCK SortInsertion
VAR_INPUT
  i_Length : INT;
END_VAR
VAR
  ix : INT;
  iy : INT;
  iz : INT;
END_VAR
VAR_IN_OUT
  ai_Data : ARRAY [0..255] OF INT;
END_VAR
VAR
  ikey : INT;
END_VAR
;
FOR ix := 1 TO i_Length-1 DO 
	ikey := ai_Data[ix];
	FOR iy := ix-1 TO 0 BY -1 DO 
		IF ai_Data[iy] > ikey THEN
			ai_Data[iy+1] := ai_Data[iy];
		ELSE
			EXIT;
		END_IF;
	END_FOR;
	ai_Data[iy+1] := ikey;
END_FOR;
END_FUNCTION_BLOCK

FUNCTION_BLOCK SortSelection
VAR_INPUT
  i_Length : INT;
END_VAR
VAR
  ix : INT;
  iy : INT;
  iz : INT;
END_VAR
VAR_IN_OUT
  ai_Data : ARRAY [0..255] OF INT;
END_VAR
VAR
  imin : INT;
END_VAR
;
FOR ix := 0 TO i_Length-2 DO 
	imin := ix;
	FOR iy := ix+1 TO i_Length-1 DO 
		IF ai_Data[iy] < ai_Data[imin] THEN
			imin := iy;
		END_IF;
	END_FOR;
	iz := ai_Data[imin];
	ai_Data[imin] := ai_Data[ix];
	ai_Data[ix] := iz;
END_FOR;
END_FUNCTION_BLOCK

FUNCTION_BLOCK ConvIP2Byte
VAR_INPUT
  dw_IP : DWORD;
END_VAR
VAR_OUTPUT
  i_Byte1 : INT;
  i_Byte2 : INT;
  i_Byte3 : INT;
  i_Byte4 : INT;
END_VAR
;
i_Byte4 := DWORD_TO_INT(dw_IP AND HFF);
i_Byte3 := DWORD_TO_INT(SHR(dw_IP, 8) AND HFF);
i_Byte2 := DWORD_TO_INT(SHR(dw_IP, 16) AND HFF);
i_Byte1 := DWORD_TO_INT(SHR(dw_IP, 24) AND HFF);
END_FUNCTION_BLOCK

FUNCTION ConvByte2IP
VAR_INPUT
  i_Byte1 : INT;
  i_Byte2 : INT;
  i_Byte3 : INT;
  i_Byte4 : INT;
END_VAR
VAR
  dw_Byte1 : DWORD;
  dw_Byte2 : DWORD;
  dw_Byte3 : DWORD;
  dw_Byte4 : DWORD;
END_VAR
;
dw_Byte1 := INT_TO_DWORD(i_Byte1) AND HFF;
dw_Byte2 := SHL(INT_TO_DWORD(i_Byte2), 8) AND HFF00;
dw_Byte3 := SHL(INT_TO_DWORD(i_Byte3), 16) AND HFF0000;
dw_Byte4 := SHL(INT_TO_DWORD(i_Byte4), 24) AND HFF000000;
ConvByte2IP := 	dw_Byte1 OR dw_Byte2 OR  dw_Byte3 OR  dw_Byte4;
END_FUNCTION

FUNCTION newSUM
VAR_INPUT
  w_IN : WORD;
END_VAR
VAR
  ix : INT;
  iy : INT;
  wTmp : WORD;
END_VAR
;
wTmp := H0001;		iy := 0;
FOR ix := 0 TO 15 DO 
	IF (wTmp AND w_IN) <> 0 THEN iy := iy + 1; END_IF;
	wTmp := SHL(wTmp,1);
END_FOR;
newSUM := iy;
END_FUNCTION

FUNCTION_BLOCK newWTOB
VAR_INPUT
  sDevNo : WORD;
  iNo : INT;
END_VAR
VAR_OUTPUT
  dDevNo : WORD;
END_VAR
VAR
  sBuffer : ARRAY [0..99] OF WORD;
  ix : INT;
  dBuffer : ARRAY [0..99] OF WORD;
END_VAR
;
BMOV(TRUE, sDevNo, iNo, sBuffer[0]); 
FOR ix := 0 TO iNo-1 DO 
		dBuffer[ix*2]		:= sBuffer[ix] AND HFF;
		dBuffer[ix*2+1]:= SHR(sBuffer[ix], 8) AND HFF;
END_FOR;
BMOV(TRUE, dBuffer[0], iNo*2, dDevNo);
END_FUNCTION_BLOCK
